TYPE T_Second : LREAL; END_TYPE

(* stored: Version 1.1.0.1, ProductVersion 3.1.4024.15
   DUT T_Second: Id {7101d999-e8a3-0210-3ae5-ad4bb8f43ba6} *)
